// TIA Portal V20 export
TYPE "LKinCtrl_PathEditor_typeHMIInterface"
// stored: Access Published
   STRUCT
      interlockID : Int;
      pathTable : "LKinCtrl_PathEditor_typePathTable";
      commandEditor : "LKinCtrl_PathEditor_typeCommandEditor";
      linkTable : "LKinCtrl_PathEditor_typeLinkTable";
   END_STRUCT;
END_TYPE
